// Mitsubishi GX Works2 project: 0708-1   PLC: Q02/Q02H

PROGRAM MAIN
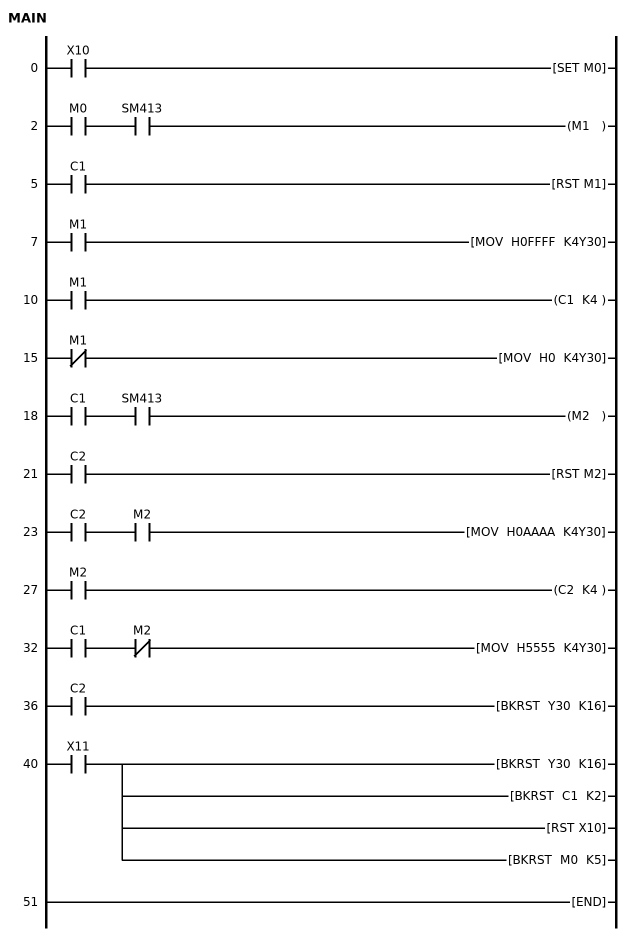
0     LD      X10
      SET     M0
2     LD      M0
      AND     SM413
      OUT     M1
5     LD      C1
      RST     M1
7     LD      M1
      MOV     H0FFFF K4Y30
10    LD      M1
      OUT     C1 K4
15    LDI     M1
      MOV     H0 K4Y30
18    LD      C1
      AND     SM413
      OUT     M2
21    LD      C2
      RST     M2
23    LD      C2
      AND     M2
      MOV     H0AAAA K4Y30
27    LD      M2
      OUT     C2 K4
32    LD      C1
      ANI     M2
      MOV     H5555 K4Y30
36    LD      C2
      BKRST   Y30 K16
40    LD      X11
      BKRST   Y30 K16
      BKRST   C1 K2
      RST     X10
      BKRST   M0 K5
51    END
END_PROGRAM
